// TIA Portal V17 export
// export: Created 2023-02-14T02:49:27.874592Z, ExportSetting WithDefaults, DisplayName Totally Integrated Automation Portal, DisplayVersion V17, DisplayName TIA Portal Openness, DisplayVersion V17, DisplayName TIA Portal Teamcenter Gateway, DisplayVersion V17, DisplayName TIA Portal Version Control Interface, DisplayVersion V17, DisplayName SINAMICS Startdrive Advanced, DisplayVersion V17, DisplayName SINAMICS Startdrive G130, G150, S120, S150, SINAMICS MV, S210, DisplayVersion V17, DisplayName SINAMICS Startdrive G110M, G120, G120C, G120D, G120P, G115D, DisplayVersion V17, DisplayName STEP 7 Professional, DisplayVersion V17, DisplayName STEP 7 Safety, DisplayVersion V17, DisplayName WinCC Professional, DisplayVersion V17
DATA_BLOCK "IO Analog Blending_DB"   // DB6
VERSION : 0.1
// stored: AutoNumber true, DBAccessibleFromOPCUA true, DBAccessibleFromWebserver true, InstanceOfName IO Analog Blending, InstanceOfType FB
"IO Analog Blending"
   // VAR_INPUT
   //    Init : Bool;
   //    Reset : Bool;
   // END_VAR
   // VAR
   //    "LT-20.01" { S7_SetPoint := 'True'} : "Ana_w_K1K2";
   //    "LT-21.01" { S7_SetPoint := 'True'} : "Ana_w_K1K2";
   //    "LT-22.01" { S7_SetPoint := 'True'} : "Ana_w_K1K2";
   //    "LT-30.01" { S7_SetPoint := 'True'} : "Ana_w_K1K2";
   //    "LT-31.01" { S7_SetPoint := 'True'} : "Ana_w_K1K2";
   //    "LT-32.01" { S7_SetPoint := 'True'} : "Ana_w_K1K2";
   //    "FT-15.01" { S7_SetPoint := 'True'} : "Ana_w_K1K2";
   //    "FT-15.01Com" { S7_SetPoint := 'True'} : "Read FT Comm";
   //    "FT-22.01" { S7_SetPoint := 'True'} : "Ana_w_K1K2";
   //    "FT-22.01Com" { S7_SetPoint := 'True'} : "Read FT Comm";
   //    "FT-32.01" { S7_SetPoint := 'True'} : "Ana_w_K1K2";
   //    "FT-32.01Com" { S7_SetPoint := 'True'} : "Read FT Comm";
   //    "LT-40.01" { S7_SetPoint := 'True'} : "Ana_w_K1K2";
   //    "LT-41.01" { S7_SetPoint := 'True'} : "Ana_w_K1K2";
   //    "FT-00.01" { S7_SetPoint := 'True'} : "Ana_w_K1K2";
   // END_VAR
BEGIN
END_DATA_BLOCK
